FUNCTION_BLOCK OUT_ANY_CONSOLE
  {SET_ATTRIBUTE(OpcUa, SERVICE)}
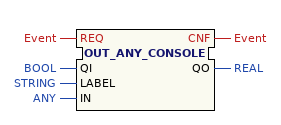
  EVENT_INPUT
    REQ;
  END_EVENT
  EVENT_OUTPUT
    CNF;
  END_EVENT
  VAR_INPUT
    QI : BOOL;
    LABEL : STRING;
    IN : ANY;
  END_VAR
  VAR_OUTPUT
    QO : REAL;
  END_VAR
END_FUNCTION_BLOCK
